// TIA Portal project "2022.09.06-编码器" (V17)

(* hardware
DEVICE "HMI_1"  KTP700 Basic PN
   slot 0: "HMI_1"  KTP700 Basic PN  6AV2 123-2GB03-0AX0  15.1.0.0
   slot 1: "HMI_RT_1"  KTP700 Basic PN  6AV2 123-2GB03-0AX0  15.1.0.0
   slot 5: "HMI_1.IE_CP_1"  PROFINET Interface  15.0.1.0
      slot 1: "PROFINET Interface_1"  PROFINET Interface
         slot 1: "Port_1"  Port
DEVICE "S7-1200 station_1"  S7-1200 Station
   slot 0: "Rack_0"  S7-1200 Rack  Rack  V1.0
   slot 1: "PLC_1"  CPU 1214C DC/DC/DC  6ES7 214-1AG40-0XB0  V4.2
*)

// ===== PLC "PLC_1"  CPU 1214C DC/DC/DC =====

VAR_GLOBAL   // PLC tag table "默认变量表"
   "启动" AT %I0.0 : Bool;
   "停止" AT %I0.1 : Bool;
   "a" AT %Q0.0 : Bool;
   "b" AT %Q0.1 : Bool;
   "c" AT %Q0.2 : Bool;
   "d" AT %Q0.3 : Bool;
   "e" AT %Q0.4 : Bool;
   "f" AT %Q0.5 : Bool;
   "g" AT %Q0.6 : Bool;
   "启动线圈" AT %M10.2 : Bool;
   "数码管显示" AT %QB0 : Byte;
   "启动按钮" AT %M10.0 : Bool;
   "停止按钮" AT %M10.1 : Bool;
END_VAR

// folder: System blocks/Program resources

DATA_BLOCK "T1-A"   // DB1
{ S7_Optimized_Access := 'TRUE' }
AUTHOR : Simatic
FAMILY : IEC
NAME : IEC_TMR
VERSION : 1.0
// stored: InstanceOfName IEC_TIMER
"IEC_TIMER"
BEGIN
END_DATA_BLOCK

DATA_BLOCK "T2-B"   // DB2
{ S7_Optimized_Access := 'TRUE' }
AUTHOR : Simatic
FAMILY : IEC
NAME : IEC_TMR
VERSION : 1.0
// stored: InstanceOfName IEC_TIMER
"IEC_TIMER"
BEGIN
END_DATA_BLOCK

DATA_BLOCK "T3-C"   // DB3
{ S7_Optimized_Access := 'TRUE' }
AUTHOR : Simatic
FAMILY : IEC
NAME : IEC_TMR
VERSION : 1.0
// stored: InstanceOfName IEC_TIMER
"IEC_TIMER"
BEGIN
END_DATA_BLOCK

DATA_BLOCK "T4_D"   // DB4
{ S7_Optimized_Access := 'TRUE' }
AUTHOR : Simatic
FAMILY : IEC
NAME : IEC_TMR
VERSION : 1.0
// stored: InstanceOfName IEC_TIMER
"IEC_TIMER"
BEGIN
END_DATA_BLOCK

DATA_BLOCK "T5-E"   // DB5
{ S7_Optimized_Access := 'TRUE' }
AUTHOR : Simatic
FAMILY : IEC
NAME : IEC_TMR
VERSION : 1.0
// stored: InstanceOfName IEC_TIMER
"IEC_TIMER"
BEGIN
END_DATA_BLOCK

DATA_BLOCK "T6-F"   // DB6
{ S7_Optimized_Access := 'TRUE' }
AUTHOR : Simatic
FAMILY : IEC
NAME : IEC_TMR
VERSION : 1.0
// stored: InstanceOfName IEC_TIMER
"IEC_TIMER"
BEGIN
END_DATA_BLOCK

DATA_BLOCK "T7-G"   // DB7
{ S7_Optimized_Access := 'TRUE' }
AUTHOR : Simatic
FAMILY : IEC
NAME : IEC_TMR
VERSION : 1.0
// stored: InstanceOfName IEC_TIMER
"IEC_TIMER"
BEGIN
END_DATA_BLOCK

DATA_BLOCK "T8-0"   // DB8
{ S7_Optimized_Access := 'TRUE' }
AUTHOR : Simatic
FAMILY : IEC
NAME : IEC_TMR
VERSION : 1.0
// stored: InstanceOfName IEC_TIMER
"IEC_TIMER"
BEGIN
END_DATA_BLOCK

DATA_BLOCK "T9-1"   // DB9
{ S7_Optimized_Access := 'TRUE' }
AUTHOR : Simatic
FAMILY : IEC
NAME : IEC_TMR
VERSION : 1.0
// stored: InstanceOfName IEC_TIMER
"IEC_TIMER"
BEGIN
END_DATA_BLOCK

DATA_BLOCK "T10-2"   // DB10
{ S7_Optimized_Access := 'TRUE' }
AUTHOR : Simatic
FAMILY : IEC
NAME : IEC_TMR
VERSION : 1.0
// stored: InstanceOfName IEC_TIMER
"IEC_TIMER"
BEGIN
END_DATA_BLOCK

DATA_BLOCK "T11-3"   // DB11
{ S7_Optimized_Access := 'TRUE' }
AUTHOR : Simatic
FAMILY : IEC
NAME : IEC_TMR
VERSION : 1.0
// stored: InstanceOfName IEC_TIMER
"IEC_TIMER"
BEGIN
END_DATA_BLOCK

DATA_BLOCK "T12-4"   // DB12
{ S7_Optimized_Access := 'TRUE' }
AUTHOR : Simatic
FAMILY : IEC
NAME : IEC_TMR
VERSION : 1.0
// stored: InstanceOfName IEC_TIMER
"IEC_TIMER"
BEGIN
END_DATA_BLOCK

DATA_BLOCK "T13-5"   // DB13
{ S7_Optimized_Access := 'TRUE' }
AUTHOR : Simatic
FAMILY : IEC
NAME : IEC_TMR
VERSION : 1.0
// stored: InstanceOfName IEC_TIMER
"IEC_TIMER"
BEGIN
END_DATA_BLOCK

DATA_BLOCK "T14-6"   // DB14
{ S7_Optimized_Access := 'TRUE' }
AUTHOR : Simatic
FAMILY : IEC
NAME : IEC_TMR
VERSION : 1.0
// stored: InstanceOfName IEC_TIMER
"IEC_TIMER"
BEGIN
END_DATA_BLOCK

DATA_BLOCK "T15-7"   // DB16
{ S7_Optimized_Access := 'TRUE' }
AUTHOR : Simatic
FAMILY : IEC
NAME : IEC_TMR
VERSION : 1.0
// stored: InstanceOfName IEC_TIMER
"IEC_TIMER"
BEGIN
END_DATA_BLOCK

DATA_BLOCK "T16-8"   // DB17
{ S7_Optimized_Access := 'TRUE' }
AUTHOR : Simatic
FAMILY : IEC
NAME : IEC_TMR
VERSION : 1.0
// stored: InstanceOfName IEC_TIMER
"IEC_TIMER"
BEGIN
END_DATA_BLOCK

DATA_BLOCK "T17-9"   // DB18
{ S7_Optimized_Access := 'TRUE' }
AUTHOR : Simatic
FAMILY : IEC
NAME : IEC_TMR
VERSION : 1.0
// stored: InstanceOfName IEC_TIMER
"IEC_TIMER"
BEGIN
END_DATA_BLOCK

DATA_BLOCK "T18-a"   // DB19
{ S7_Optimized_Access := 'TRUE' }
AUTHOR : Simatic
FAMILY : IEC
NAME : IEC_TMR
VERSION : 1.0
// stored: InstanceOfName IEC_TIMER
"IEC_TIMER"
BEGIN
END_DATA_BLOCK

DATA_BLOCK "T19-b"   // DB20
{ S7_Optimized_Access := 'TRUE' }
AUTHOR : Simatic
FAMILY : IEC
NAME : IEC_TMR
VERSION : 1.0
// stored: InstanceOfName IEC_TIMER
"IEC_TIMER"
BEGIN
END_DATA_BLOCK

DATA_BLOCK "T20-C"   // DB21
{ S7_Optimized_Access := 'TRUE' }
AUTHOR : Simatic
FAMILY : IEC
NAME : IEC_TMR
VERSION : 1.0
// stored: InstanceOfName IEC_TIMER
"IEC_TIMER"
BEGIN
END_DATA_BLOCK

DATA_BLOCK "T21-d"   // DB22
{ S7_Optimized_Access := 'TRUE' }
AUTHOR : Simatic
FAMILY : IEC
NAME : IEC_TMR
VERSION : 1.0
// stored: InstanceOfName IEC_TIMER
"IEC_TIMER"
BEGIN
END_DATA_BLOCK

DATA_BLOCK "T22-e"   // DB23
{ S7_Optimized_Access := 'TRUE' }
AUTHOR : Simatic
FAMILY : IEC
NAME : IEC_TMR
VERSION : 1.0
// stored: InstanceOfName IEC_TIMER
"IEC_TIMER"
BEGIN
END_DATA_BLOCK

DATA_BLOCK "T23-f"   // DB24
{ S7_Optimized_Access := 'TRUE' }
AUTHOR : Simatic
FAMILY : IEC
NAME : IEC_TMR
VERSION : 1.0
// stored: InstanceOfName IEC_TIMER
"IEC_TIMER"
BEGIN
END_DATA_BLOCK

// folder: (top level)

ORGANIZATION_BLOCK "Main"   // OB1, LAD, ProgramCycle
TITLE = "Main Program Sweep (Cycle)"
{ S7_Optimized_Access := 'TRUE' }
VERSION : 0.1
   VAR_INPUT
      Initial_Call : Bool;   // Initial call of this OB
      Remanence : Bool;   // =True, if remanent data are available
   END_VAR
BEGIN

REGION Network 1
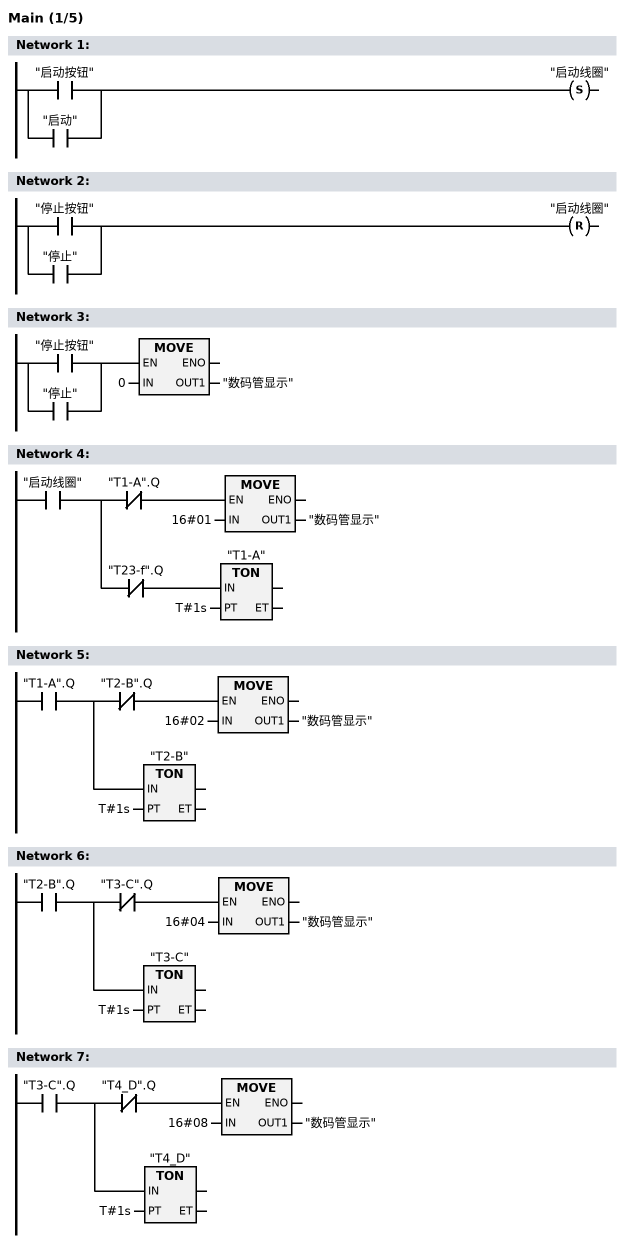
   RUNG wire#powerrail
      Contact( "启动按钮" )
      wire#w1
      S_Coil( "启动线圈" )
   END_RUNG
   RUNG wire#powerrail
      Contact( "启动" )
   END_RUNG wire#w1
   // the same network as SCL:
   IF "启动按钮" OR "启动" THEN "启动线圈" := TRUE; END_IF;
END_REGION

REGION Network 2
   RUNG wire#powerrail
      Contact( "停止按钮" )
      wire#w1
      R_Coil( "启动线圈" )
   END_RUNG
   RUNG wire#powerrail
      Contact( "停止" )
   END_RUNG wire#w1
   // the same network as SCL:
   IF "停止按钮" OR "停止" THEN "启动线圈" := FALSE; END_IF;
END_REGION

REGION Network 3
   RUNG wire#powerrail
      Contact( "停止按钮" )
      wire#w1
      Move(in := 0, out1 => "数码管显示")
   END_RUNG
   RUNG wire#powerrail
      Contact( "停止" )
   END_RUNG wire#w1
   // the same network as SCL:
   IF "停止按钮" OR "停止" THEN "数码管显示" := 0; END_IF;
END_REGION

REGION Network 4
   IF "启动线圈" AND NOT "T1-A".Q THEN "数码管显示" := 16#01; END_IF;
   "T1-A".TON(IN := "启动线圈" AND NOT "T23-f".Q, PT := T#1s);
END_REGION

REGION Network 5
   IF "T1-A".Q AND NOT "T2-B".Q THEN "数码管显示" := 16#02; END_IF;
   "T2-B".TON(IN := "T1-A".Q, PT := T#1s);
END_REGION

REGION Network 6
   IF "T2-B".Q AND NOT "T3-C".Q THEN "数码管显示" := 16#04; END_IF;
   "T3-C".TON(IN := "T2-B".Q, PT := T#1s);
END_REGION

REGION Network 7
   IF "T3-C".Q AND NOT "T4_D".Q THEN "数码管显示" := 16#08; END_IF;
   "T4_D".TON(IN := "T3-C".Q, PT := T#1s);
END_REGION

REGION Network 8
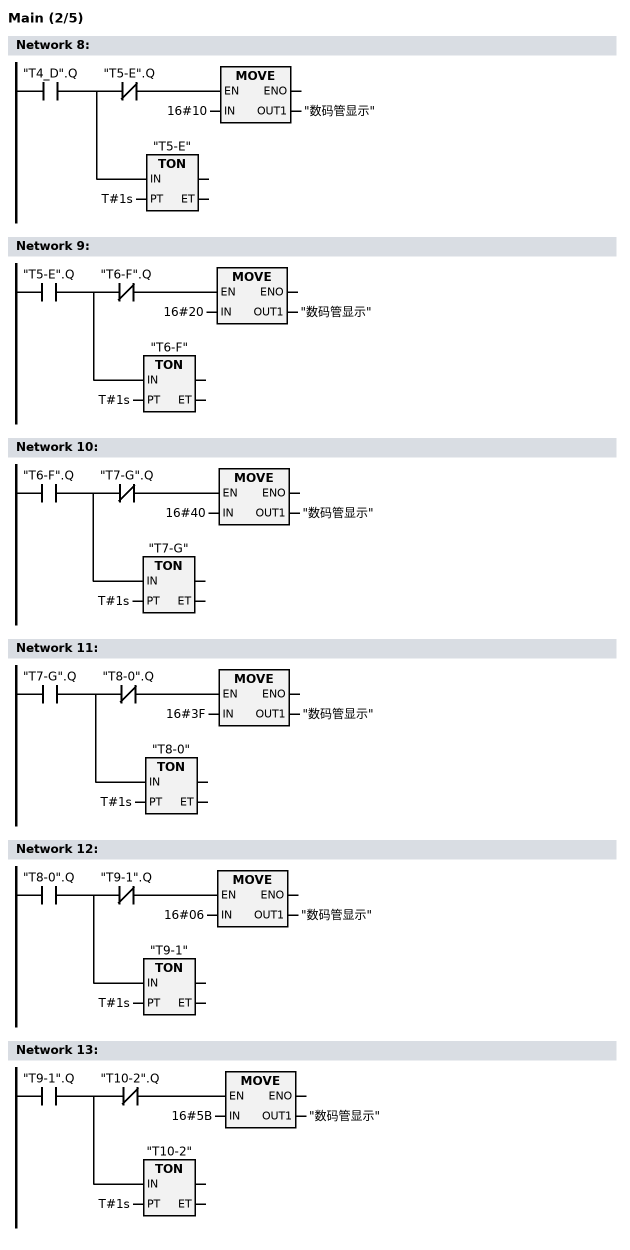
   IF "T4_D".Q AND NOT "T5-E".Q THEN "数码管显示" := 16#10; END_IF;
   "T5-E".TON(IN := "T4_D".Q, PT := T#1s);
END_REGION

REGION Network 9
   IF "T5-E".Q AND NOT "T6-F".Q THEN "数码管显示" := 16#20; END_IF;
   "T6-F".TON(IN := "T5-E".Q, PT := T#1s);
END_REGION

REGION Network 10
   IF "T6-F".Q AND NOT "T7-G".Q THEN "数码管显示" := 16#40; END_IF;
   "T7-G".TON(IN := "T6-F".Q, PT := T#1s);
END_REGION

REGION Network 11
   IF "T7-G".Q AND NOT "T8-0".Q THEN "数码管显示" := 16#3F; END_IF;
   "T8-0".TON(IN := "T7-G".Q, PT := T#1s);
END_REGION

REGION Network 12
   IF "T8-0".Q AND NOT "T9-1".Q THEN "数码管显示" := 16#06; END_IF;
   "T9-1".TON(IN := "T8-0".Q, PT := T#1s);
END_REGION

REGION Network 13
   IF "T9-1".Q AND NOT "T10-2".Q THEN "数码管显示" := 16#5B; END_IF;
   "T10-2".TON(IN := "T9-1".Q, PT := T#1s);
END_REGION

REGION Network 14
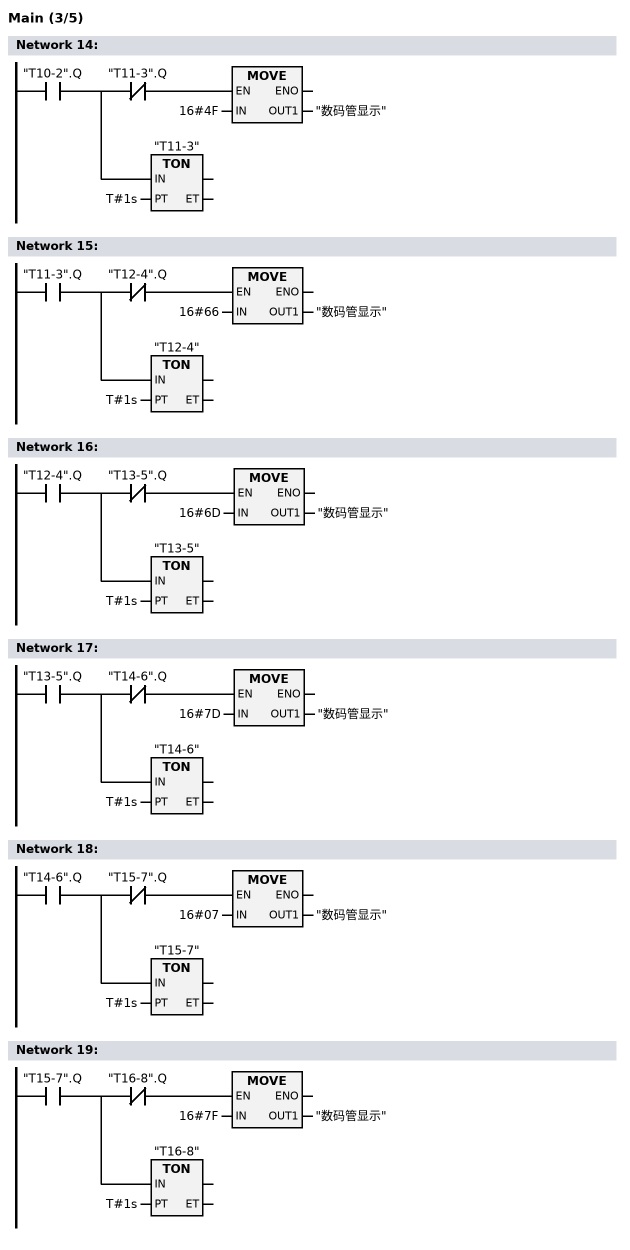
   IF "T10-2".Q AND NOT "T11-3".Q THEN "数码管显示" := 16#4F; END_IF;
   "T11-3".TON(IN := "T10-2".Q, PT := T#1s);
END_REGION

REGION Network 15
   IF "T11-3".Q AND NOT "T12-4".Q THEN "数码管显示" := 16#66; END_IF;
   "T12-4".TON(IN := "T11-3".Q, PT := T#1s);
END_REGION

REGION Network 16
   IF "T12-4".Q AND NOT "T13-5".Q THEN "数码管显示" := 16#6D; END_IF;
   "T13-5".TON(IN := "T12-4".Q, PT := T#1s);
END_REGION

REGION Network 17
   IF "T13-5".Q AND NOT "T14-6".Q THEN "数码管显示" := 16#7D; END_IF;
   "T14-6".TON(IN := "T13-5".Q, PT := T#1s);
END_REGION

REGION Network 18
   IF "T14-6".Q AND NOT "T15-7".Q THEN "数码管显示" := 16#07; END_IF;
   "T15-7".TON(IN := "T14-6".Q, PT := T#1s);
END_REGION

REGION Network 19
   IF "T15-7".Q AND NOT "T16-8".Q THEN "数码管显示" := 16#7F; END_IF;
   "T16-8".TON(IN := "T15-7".Q, PT := T#1s);
END_REGION

REGION Network 20
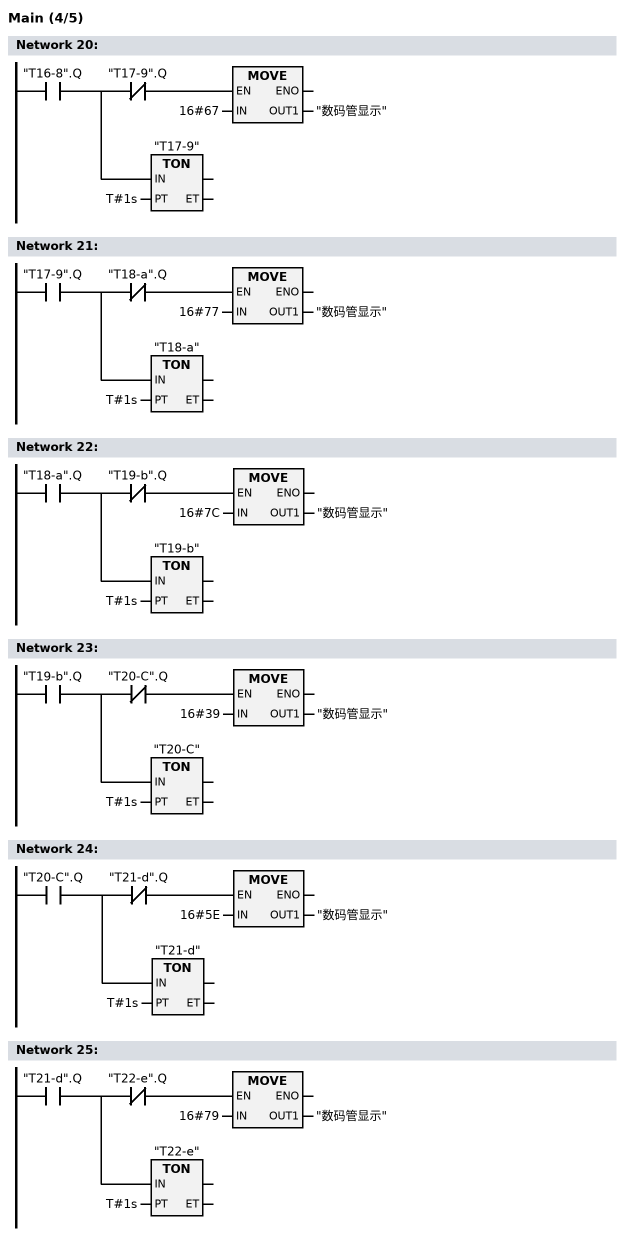
   IF "T16-8".Q AND NOT "T17-9".Q THEN "数码管显示" := 16#67; END_IF;
   "T17-9".TON(IN := "T16-8".Q, PT := T#1s);
END_REGION

REGION Network 21
   IF "T17-9".Q AND NOT "T18-a".Q THEN "数码管显示" := 16#77; END_IF;
   "T18-a".TON(IN := "T17-9".Q, PT := T#1s);
END_REGION

REGION Network 22
   IF "T18-a".Q AND NOT "T19-b".Q THEN "数码管显示" := 16#7C; END_IF;
   "T19-b".TON(IN := "T18-a".Q, PT := T#1s);
END_REGION

REGION Network 23
   IF "T19-b".Q AND NOT "T20-C".Q THEN "数码管显示" := 16#39; END_IF;
   "T20-C".TON(IN := "T19-b".Q, PT := T#1s);
END_REGION

REGION Network 24
   IF "T20-C".Q AND NOT "T21-d".Q THEN "数码管显示" := 16#5E; END_IF;
   "T21-d".TON(IN := "T20-C".Q, PT := T#1s);
END_REGION

REGION Network 25
   IF "T21-d".Q AND NOT "T22-e".Q THEN "数码管显示" := 16#79; END_IF;
   "T22-e".TON(IN := "T21-d".Q, PT := T#1s);
END_REGION

REGION Network 26
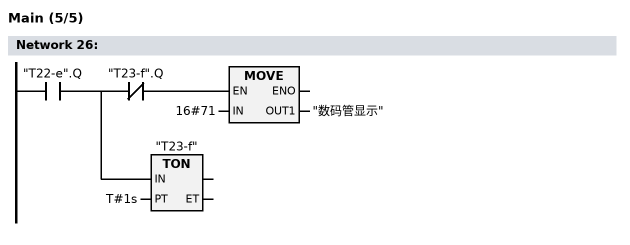
   IF "T22-e".Q AND NOT "T23-f".Q THEN "数码管显示" := 16#71; END_IF;
   "T23-f".TON(IN := "T22-e".Q, PT := T#1s);
END_REGION
END_ORGANIZATION_BLOCK

(* ===== HMI "HMI_RT_1" =====
system functions are stored by id; their names below are inferred from use
connection "HMI_连接_1": ETHERNET, SMART_S7_1200_OMS

HMI tags "默认变量表"
   "启动按钮" : Bool = PLC 启动按钮 AT %M10.0, 1 s
   "停止按钮" : Bool = PLC 停止按钮 AT %M10.1, 1 s
   "a" : Bool = PLC a AT %Q0.0, 1 s
   "b" : Bool = PLC b AT %Q0.1, 1 s
   "c" : Bool = PLC c AT %Q0.2, 1 s
   "d" : Bool = PLC d AT %Q0.3, 1 s
   "e" : Bool = PLC e AT %Q0.4, 1 s
   "f" : Bool = PLC f AT %Q0.5, 1 s
   "g" : Bool = PLC g AT %Q0.6, 1 s

screen "画面_1" 800x480
   Rectangle "矩形_1" at 590,157 size 118x19
      Appearance <- "a"
   Rectangle "矩形_2" at 591,251 size 118x19
      Appearance <- "g"
   Rectangle "矩形_3" at 593,345 size 118x19
      Appearance <- "d"
   Rectangle "矩形_4" at 712,174 size 19x75
      Appearance <- "b"
   Rectangle "矩形_5" at 570,270 size 19x75
      Appearance <- "e"
   Rectangle "矩形_6" at 713,268 size 19x75
      Appearance <- "c"
   Rectangle "矩形_7" at 569,177 size 19x75
      Appearance <- "f"
   Button "按钮_1" at 421,198 size 96x32; TextOff '启动'
      on Press: SetBit("启动按钮")
      on Release: ResetBit("启动按钮")
   Button "按钮_2" at 421,293 size 96x32; TextOff '停止'
      on Release: ResetBit("停止按钮")
      on Press: SetBit("停止按钮")
*)